// SIMATIC S7-200 project (STEP 7-Micro/WIN), CPU 224XP CN REL 02.01

ORGANIZATION_BLOCK 主程序:OB1
TITLE=程序注释
BEGIN
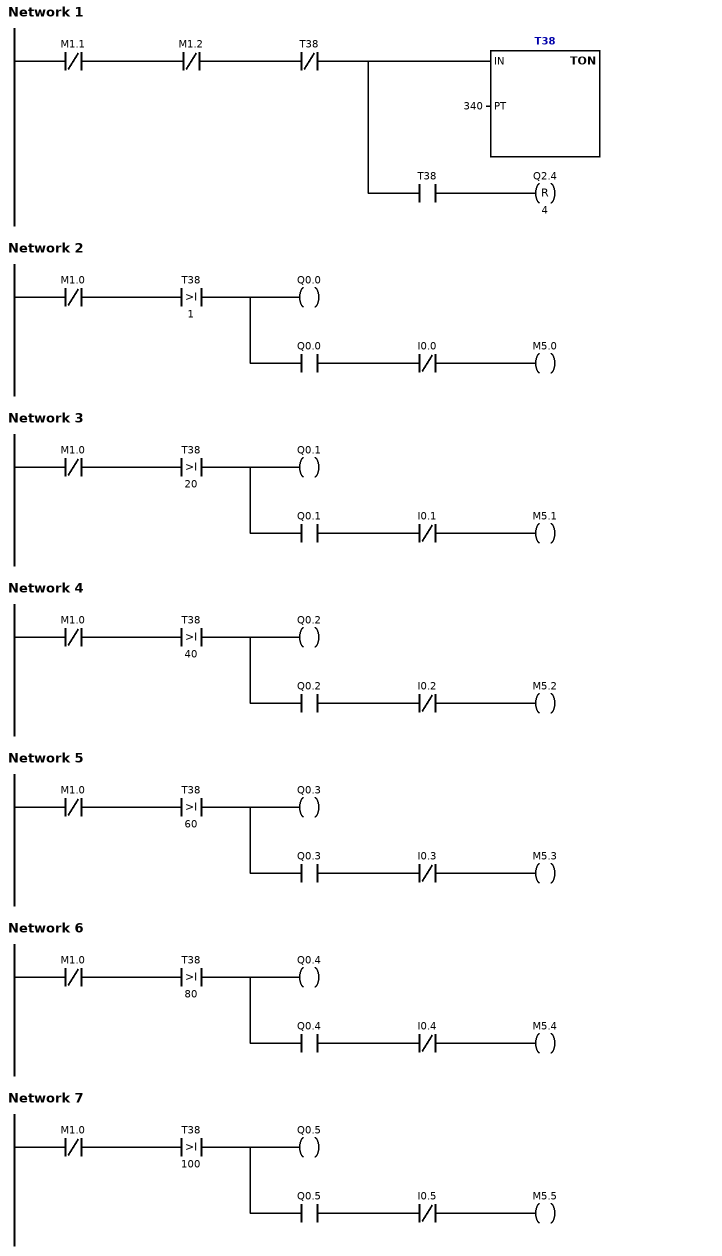
Network 1
LDN    M1.1
AN     M1.2
AN     T38
TON    T38, 340
A      T38
R      Q2.4, 4
Network 2
LDN    M1.0
AW>    T38, 1
=      Q0.0
A      Q0.0
AN     I0.0
=      M5.0
Network 3
LDN    M1.0
AW>    T38, 20
=      Q0.1
A      Q0.1
AN     I0.1
=      M5.1
Network 4
LDN    M1.0
AW>    T38, 40
=      Q0.2
A      Q0.2
AN     I0.2
=      M5.2
Network 5
LDN    M1.0
AW>    T38, 60
=      Q0.3
A      Q0.3
AN     I0.3
=      M5.3
Network 6
LDN    M1.0
AW>    T38, 80
=      Q0.4
A      Q0.4
AN     I0.4
=      M5.4
Network 7
LDN    M1.0
AW>    T38, 100
=      Q0.5
A      Q0.5
AN     I0.5
=      M5.5
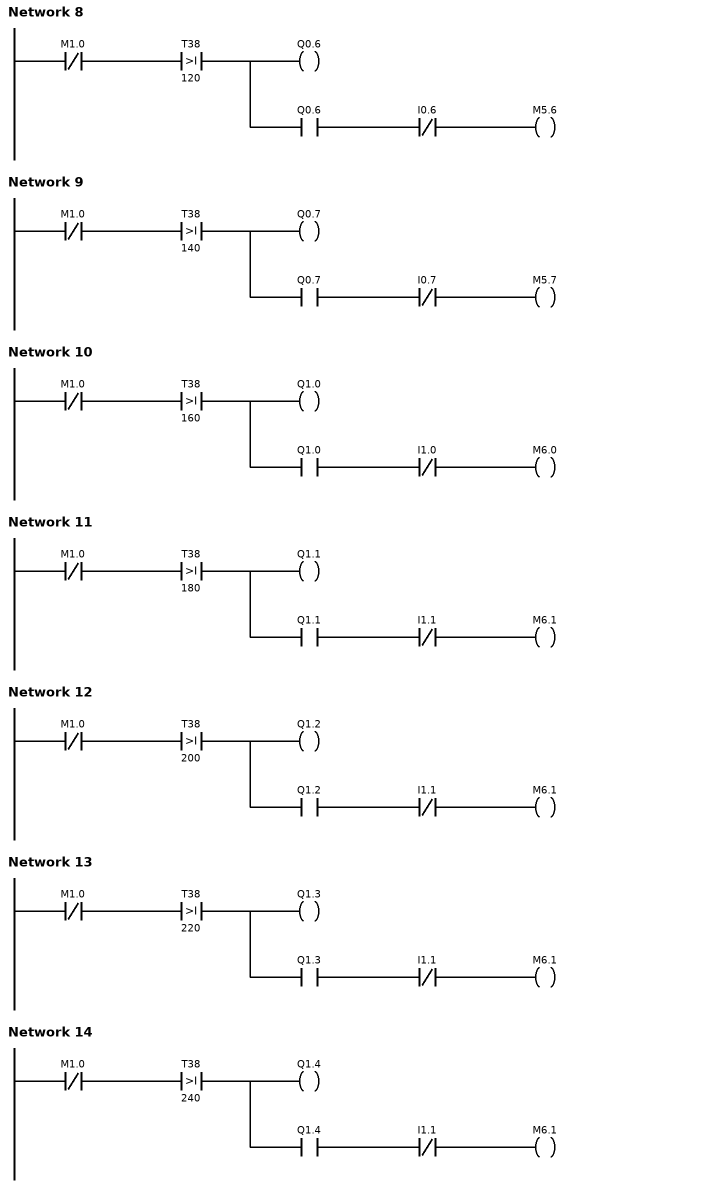
Network 8
LDN    M1.0
AW>    T38, 120
=      Q0.6
A      Q0.6
AN     I0.6
=      M5.6
Network 9
LDN    M1.0
AW>    T38, 140
=      Q0.7
A      Q0.7
AN     I0.7
=      M5.7
Network 10
LDN    M1.0
AW>    T38, 160
=      Q1.0
A      Q1.0
AN     I1.0
=      M6.0
Network 11
LDN    M1.0
AW>    T38, 180
=      Q1.1
A      Q1.1
AN     I1.1
=      M6.1
Network 12
LDN    M1.0
AW>    T38, 200
=      Q1.2
A      Q1.2
AN     I1.1
=      M6.1
Network 13
LDN    M1.0
AW>    T38, 220
=      Q1.3
A      Q1.3
AN     I1.1
=      M6.1
Network 14
LDN    M1.0
AW>    T38, 240
=      Q1.4
A      Q1.4
AN     I1.1
=      M6.1
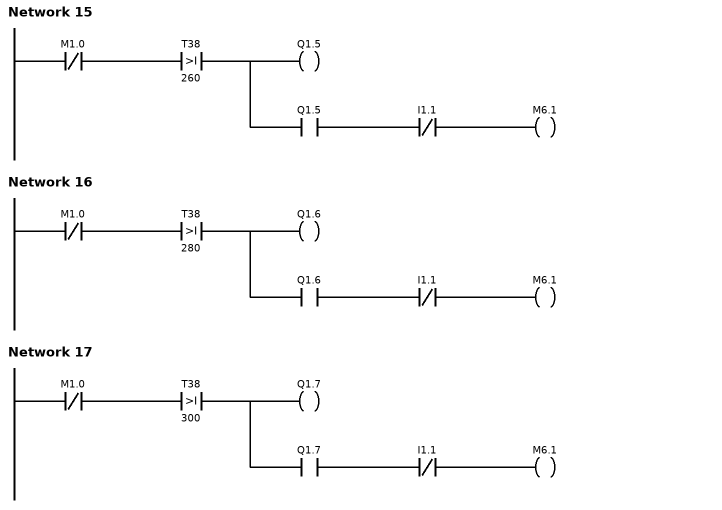
Network 15
LDN    M1.0
AW>    T38, 260
=      Q1.5
A      Q1.5
AN     I1.1
=      M6.1
Network 16
LDN    M1.0
AW>    T38, 280
=      Q1.6
A      Q1.6
AN     I1.1
=      M6.1
Network 17
LDN    M1.0
AW>    T38, 300
=      Q1.7
A      Q1.7
AN     I1.1
=      M6.1
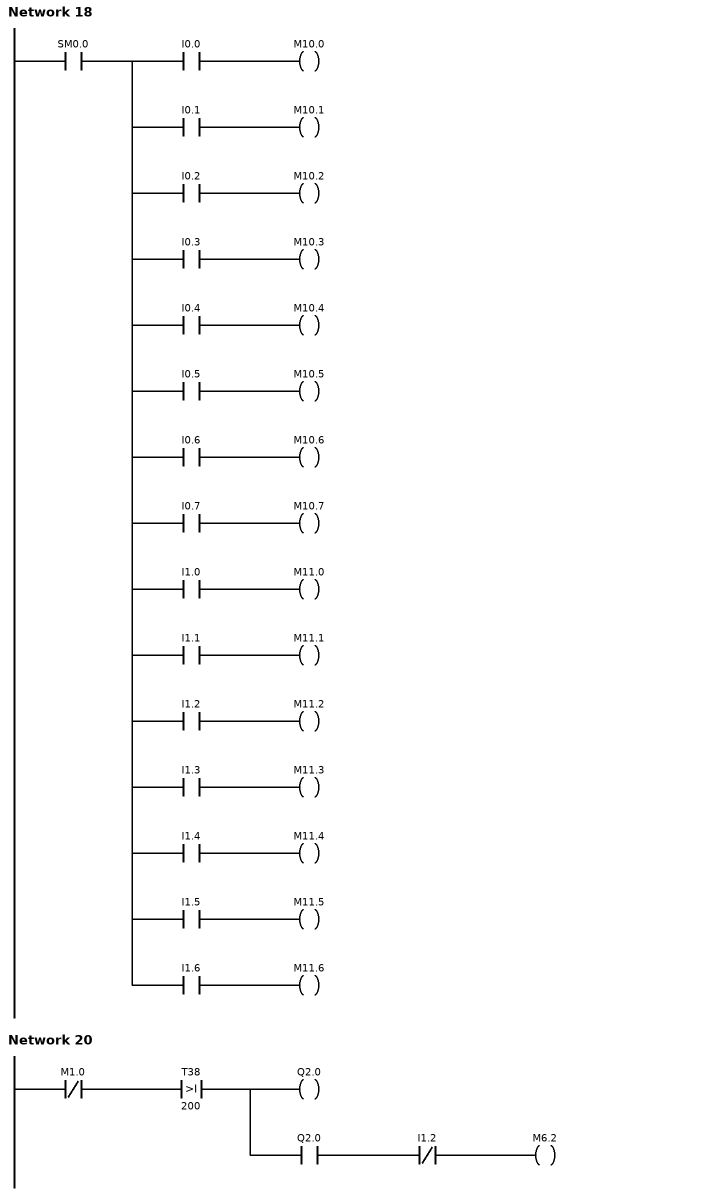
Network 18
// (network saved uncompiled; LAD cells follow)
// row 0: c0 -| |- SM0.0 v  c1 -| |- I0.0  c2 -( ) M10.0
// row 1: c0 ^v  c1 -| |- I0.1  c2 -( ) M10.1
// row 2: c0 ^v  c1 -| |- I0.2  c2 -( ) M10.2
// row 3: c0 ^v  c1 -| |- I0.3  c2 -( ) M10.3
// row 4: c0 ^v  c1 -| |- I0.4  c2 -( ) M10.4
// row 5: c0 ^v  c1 -| |- I0.5  c2 -( ) M10.5
// row 6: c0 ^v  c1 -| |- I0.6  c2 -( ) M10.6
// row 7: c0 ^v  c1 -| |- I0.7  c2 -( ) M10.7
// row 8: c0 ^v  c1 -| |- I1.0  c2 -( ) M11.0
// row 9: c0 ^v  c1 -| |- I1.1  c2 -( ) M11.1
// row 10: c0 ^v  c1 -| |- I1.2  c2 -( ) M11.2
// row 11: c0 ^v  c1 -| |- I1.3  c2 -( ) M11.3
// row 12: c0 ^v  c1 -| |- I1.4  c2 -( ) M11.4
// row 13: c0 ^v  c1 -| |- I1.5  c2 -( ) M11.5
// row 14: c0 ^  c1 -| |- I1.6  c2 -( ) M11.6
Network 20
LDN    M1.0
AW>    T38, 200
=      Q2.0
A      Q2.0
AN     I1.2
=      M6.2
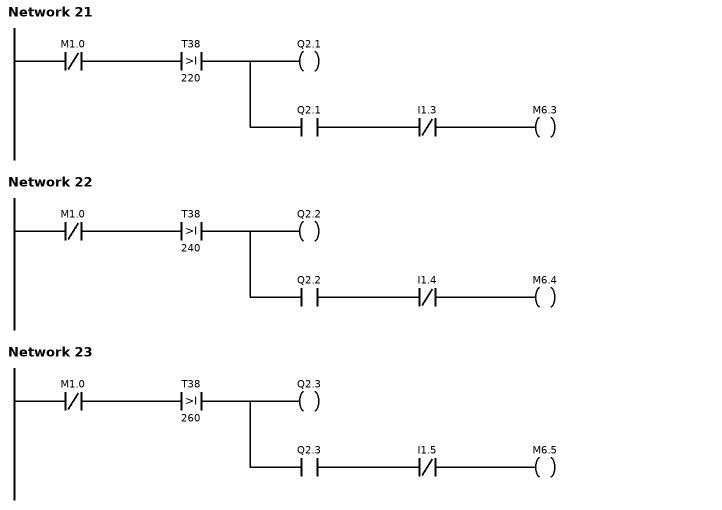
Network 21
LDN    M1.0
AW>    T38, 220
=      Q2.1
A      Q2.1
AN     I1.3
=      M6.3
Network 22
LDN    M1.0
AW>    T38, 240
=      Q2.2
A      Q2.2
AN     I1.4
=      M6.4
Network 23
LDN    M1.0
AW>    T38, 260
=      Q2.3
A      Q2.3
AN     I1.5
=      M6.5
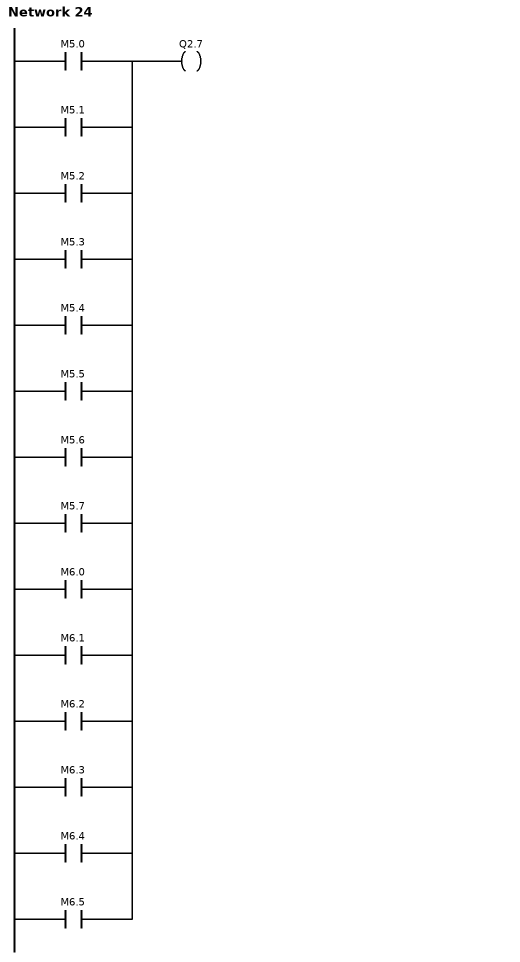
Network 24
LD     M5.0
O      M5.1
O      M5.2
O      M5.3
O      M5.4
O      M5.5
O      M5.6
O      M5.7
O      M6.0
O      M6.1
O      M6.2
O      M6.3
O      M6.4
O      M6.5
=      Q2.7
END_ORGANIZATION_BLOCK
